FUNCTION_BLOCK FB_HydMixCir
VAR_INPUT
	//Pump
	iPump			:	I_Pump;
	//Valve
	iValve			:	I_Valve;
	//Temperatures
	iTempSupPrim	:	I_TemperatureSensor;
	iTempRetPrim	:	I_TemperatureSensor;
	iTempSup		:	I_TemperatureSensor;
	iTempRet		:	I_TemperatureSensor;
	//Controller
	iControl		:	I_HydraulicMixingControl;
END_VAR
VAR_OUTPUT
END_VAR
VAR
	eMode : E_ControlMode := E_ControlMode.Off;
END_VAR

PROPERTY Mode : E_ControlMode
GET
Mode := THIS^.eMode;
END_GET
SET
THIS^.eMode := Mode;
END_SET
END_PROPERTY

METHOD Run
VAR_INPUT
END_VAR
//Update temperatures
iTempSupPrim.Run();
iTempRetPrim.Run();
iTempSup.Run();
iTempRet.Run();

//Run components
iPump.Run();
iValve.Run();

//Run controller
iControl.Mode := eMode;
iControl.TemperatureSupAct := iTempSup.Temperature;
iControl.Run();

//Pump set properties
IF eMode = E_ControlMode.Off THEN
	iPump.SetOn := FALSE;
ELSE
	iPump.SetOn := TRUE;
END_IF
iPump.ControlMode := iControl.PumpMode;
iPump.Setpoint := iControl.PumpSet;

//Valve set properties
iValve.OpeningSetpoint := iControl.ValveSet;
END_METHOD

END_FUNCTION_BLOCK

(* stored: Version 1.1.0.1, ProductVersion 3.1.4024.3
   POU FB_HydMixCir: Id {bf69e14a-3468-49db-9e18-f972a718c19a}, SpecialFunc None
   Property Mode: Id {70e12eae-b206-485e-83ad-672f3b39b70b}
   Get Get: Id {2bbe612f-3140-48f7-b2ad-c7901abcc897}
   Set Set: Id {d6e6093c-70de-4d6b-b7e6-96e291088501}
   Method Run: Id {11164a5a-f7c1-43f5-8f73-4ba44b0ac571} *)
